TEXTLIST TextList_00
   = ''
END_TEXTLIST

(* stored: Version 1.1.0.1
   TextList TextList_00: Id {125067f5-fc8c-061f-31cc-342479ef7f05} *)
